TYPE PriceItem : 
STRUCT 
	price : REAL;
	index : INT; 
END_STRUCT 
END_TYPE

(* stored: Version 1.1.0.1
   DUT PriceItem: Id {38e70dbd-aaa4-4ff1-8c51-9a60acc7ff88} *)
